{attribute 'GeneratedUsingTerminal: EJ6002-0000-0016'}
{attribute addProperty BoxType "EJ6002-0000-0016"}
{attribute addProperty Id "StatusAT %I*Status_3D84275F8Data_InAT %I*ARRAY[0..21] OF USINT22"}
{attribute addProperty CRC "1334739266"}
{attribute addProperty Size "30"}
TYPE COM_Inputs_Channel_3801C95E :
STRUCT
	{attribute addProperty Name "Status"}
	Status AT %I* : Status_3D84275F;
	{attribute addProperty Name "Data_In"}
	Data_In AT %I* : ARRAY[0..21] OF USINT;
END_STRUCT
END_TYPE

(* stored: Version 1.2.0.0, ProductVersion 3.1.4024.9
   DUT COM_Inputs_Channel_3801C95E: Id {788863ac-4fd7-48ff-bdf6-e8f91c97187c} *)
